(* CODESYS project GomelChemical.export

Project tree, tasks and I/O mapping:
  application Application
    libraries: 
    task PLC_Task (cyclic, interval t#50ms, priority 15) calls PLC_PRG
    GV/
      global variables _DO
      global variables AI
      global variables AO
      global variables DI
      global variables Hard
      global variables HMI_Sensors
      global variables HMI_Setting
    IO/
      function AI_TO_Current [ST]
      program prAItoValue [ST]
      program prInToVars [ST]
      program prVarsToOut [ST]
    program PLC_PRG [ST]
*)

// Application/GV/_DO

VAR_GLOBAL
	DO_SupplyStart_57_1	: BOOL;
	DO_SupplyStop_57_1	: BOOL;
	DO_SupplyStart_57_2	: BOOL;
	DO_SupplyStop_57_2	: BOOL;
	DO_SupplyStart_71_1	: BOOL;
	DO_SupplyStop_71_1	: BOOL;
	DO_SupplyStart_71_2	: BOOL;
	DO_SupplyStop_71_2	: BOOL;
	DO_SupplyStart_81_1	: BOOL;
	DO_SupplyStop_81_1	: BOOL;
	DO_MaxLevel_70_1_70_2_Stp_Elv8_Cvr5_6A:	BOOL;
	DO_MaxLevel_86_Stp_Elv8_Cvr5_7:	BOOL;
	DO_MinLevel_49_Stp_Pump_50:	BOOL;
	DO_MaxLevel_49_Stp_Pump_50:	BOOL;
	DO_MinLevel_67_Stp_Pump_68:	BOOL;
	DO_MaxLevel_67_Stp_Pump_68:	BOOL;
	DO_MinLevel_67_Stp_Pump_68_1:	BOOL;
	DO_MaxLevel_67_Stp_Pump_68_1:	BOOL;
	DO_MinLevel_103_1_Stp_Pump_103_1A:	BOOL;
	DO_MinLevelL1_103_1_Stp_Pump_103_1B:	BOOL;
	DO_MinLevelL2_103_1_Stp_Pump_103_1B:	BOOL;
	
//////////////////////////////////////////////////////////////////////	
	
	_DO_SupplyStart_57_1	: BOOL;
	_DO_SupplyStop_57_1	: BOOL;
	_DO_SupplyStart_57_2	: BOOL;
	_DO_SupplyStop_57_2	: BOOL;
	_DO_SupplyStart_71_1	: BOOL;
	_DO_SupplyStop_71_1	: BOOL;
	_DO_SupplyStart_71_2	: BOOL;
	_DO_SupplyStop_71_2	: BOOL;
	_DO_SupplyStart_81_1	: BOOL;
	_DO_SupplyStop_81_1	: BOOL;
	_DO_MaxLevel_70_1_70_2_Stp_Elv8_Cvr5_6A:	BOOL;
	_DO_MaxLevel_86_Stp_Elv8_Cvr5_7:	BOOL;
	_DO_MinLevel_49_Stp_Pump_50:	BOOL;
	_DO_MaxLevel_49_Stp_Pump_50:	BOOL;
	_DO_MinLevel_67_Stp_Pump_68:	BOOL;
	_DO_MaxLevel_67_Stp_Pump_68:	BOOL;
	_DO_MinLevel_67_Stp_Pump_68_1:	BOOL;
	_DO_MaxLevel_67_Stp_Pump_68_1:	BOOL;
	_DO_MinLevel_103_1_Stp_Pump_103_1A:	BOOL;
	_DO_MinLevelL1_103_1_Stp_Pump_103_1B:	BOOL;
	_DO_MinLevelL2_103_1_Stp_Pump_103_1B:	BOOL;
	
	
END_VAR

// Application/GV/AI

VAR_GLOBAL
	AI_TgasBeforeDryerDrum_45		: INT;
	AI_TgasAfterDryerDrum_45		: INT;
	AI_TgasFurnace_120				: INT;
	AI_TproductAfterDryerDrum_45	: INT;
	AI_TairCooler					: INT;
	AI_TairAfterDrumCond_76			: INT;
	AI_Tvent_53_3_1					: INT;
	AI_Tvent_53_3_2					: INT;
	AI_Tvent_53_2_1					: INT;
	AI_Tvent_53_2_2					: INT;
	AI_Tvent_53_1_1					: INT;
	AI_Tvent_53_1_2					: INT;
	
	AI_Tvent_65_0_1					: INT;
	AI_Tvent_65_0_2					: INT;
	AI_Tvent_65_1_1					: INT;
	AI_Tvent_65_1_2					: INT;
	AI_Tvent_65_2_1					: INT;
	AI_Tvent_65_2_2					: INT;
	AI_Tretur_61					: INT;
	AI_Ttank_103_1					: INT;
	AI_AirPressureBeforeBurner		: INT;
	AI_AirFirstPressureBeforeFurnace_120		: INT;
	AI_AirSecondPressureBeforeFurnace_120		: INT;
	AI_PCV22Pos						: INT;
	AI_UnderPresFurnace_120			: INT;
	AI_UnderPresGranul_31			: INT;
	AI_UnderPresDryerDrum_45		: INT;
	AI_UnderPresCooler_63_1			: INT;
	AI_PressureKiPA					: INT;
	AI_UnderPresBeforeAbsorbAKT_37	: INT;
	AI_UnderPresAfterAbsorbAKT_37	: INT;
	AI_UnderPresAfterAPS_48			: INT;
	AI_UnderPresBeforeHydroCycl_21	: INT;
	AI_UnderPresAfterHydroCycl_21	: INT;
	AI_UnderPresSalex_211			: INT;
	AI_AbsorbConsumInHydroCycl_21	: INT;
	AI_AbsorbConsumBeforeHydroCycl_21	: INT;
	AI_GasConsumBeforeBurner		: INT;
	AI_FCV16Pos						: INT;
	AI_AirConsumeFurnace_120		: INT;
	AI_FCV18Pos						: INT;
	AI_ReturConsumGranul_31			: INT;
	AI_AbsorLiquidConsumbAKT_37_FT100		: INT;
	AI_WaterConsumAbsorbSystem		: INT;
	AI_AbsorLiquidScuber_66_12		: INT;
	AI_AbsorLiquidTank_103_1		: INT;
	AI_FCV113						: INT;
	AI_ConsumBeforeScrubber_66_1	: INT;
	AI_ConsumInAPS_48				: INT;
	AI_ConsumH2SO4_102_to_35		: INT;
	AI_ConsumH2SO4_102_to_103		: INT;
	AI_AbsorLiquidConsumbAKT_37_FT132		: INT;
	AI_Consum_H3PO4					: INT;
	AI_ConsumH2SO4					: INT;
	AI_ConsumPressedAirToZech		: INT;
	AI_ConsumPressedAir				: INT;
	AI_ConsumChlKToGran_FQUIR_12_31	: INT;
	AI_ConsumKarbanToGran_31		: INT;
	AI_ConsumChlKToGran_FQUIR_17_31	: INT;
	AI_ConsumMicroAddToGran_31_FQUIR_57_1	: INT;
	AI_ConsumMicroAddToGran_31_FQUIR_57_2	: INT;
	AI_OilLevel_78					: INT;
	AI_CycleTankLevel_49			: INT;
	AI_LCV101Pos					: INT;
	AI_CollectorTankLevel_35		: INT;
	AI_CycleTankLevel_67			: INT;
	AI_CollectorTankLevel_103_1		: INT;
	AI_ReceivTankH3PO4level_41		: INT;
	AI_ReceivTankH3PO4level_39		: INT;
	AI_SupplyTankH3PO4level_25		: INT;
	AI_LCV203Pos					: INT;
	AI_TankH2SO4Level_102			: INT;
	AI_SupplyTankH2SO4Level_102_a	: INT;
	AI_LCV206Pos					: INT;
	AI_pH_CollectorTank_35			: INT;
	AI_ACV104Pos					: INT;
	AI_pH_CyclTank_49				: INT;
	AI_ACV112Pos					: INT;
	AI_pH_CollectorTank_103_1		: INT;
	AI_ACV115Pos					: INT;
	AI_OutAirWetness				: INT;
	AI_DryerRoomAirWetness_45			: INT;
	AI_IssuedProductWeight_203			: INT;
	AI_TubeReactorTemp_100_TE9			: INT;
	AI_AntiCackTempInReceiveTank_81	: INT;
	AI_TCV302Pos					: INT;
	AI_AntiCackTempInSupplyTank_81_TT303	: INT;
	AI_TCV303Pos					: INT;
	AI_TubeReactorTemp_100_TE304	: INT;
	AI_H2SO4_PressureBeforeTubeReactor_100	: INT;
	AI_H3PO4_PressureBeforeTubeReactor_100	: INT;
	AI_AcidWaistPressure_100				: INT;
	AI_H2SO4_PressureBeforeTubeReactor_100_1	: INT;
	AI_H3PO4_PressureBeforeTubeReactor_100_1	: INT;
	AI_AcidWaistPressure_100_1				: INT;
	AI_H2SO4ConsumTubeReactor_100		: INT;
	AI_FCV3Pos					: INT;
	AI_H3PO4ConsumTubeReactor_100		: INT;
	AI_FCV4Pos					: INT;
	AI_AcidWaistConsume_100				: INT;
	AI_FCV5Pos					: INT;
	AI_FCV10Pos					: INT;
	AI_FCV214Pos					: INT;
	AI_FCV341Pos					: INT;
	AI_FCV342Pos					: INT;
	AI_H2SO4ConsumTubeReactor_100_1		: INT;
	AI_FCV343Pos					: INT;
	AI_H3PO4ConsumTubeReactor_100_1		: INT;
	AI_FCV344Pos					: INT;
	AI_AcidWaistConsume_100_1		: INT;
	AI_FCV345Pos					: INT;
	AI_FCV346Pos					: INT;
	AI_AntiCackLevelInReceivTank_81	: INT;
	AI_AntiCackLevelInSupplyTank_82	: INT;
	AI_SubPumpCurrent_102_B				: INT;
	AI_SubPumpCurrent_103_1B		: INT;
	
	
	
	//////////////////////////////////////////////////////////////////
	
	_AI_TgasBeforeDryerDrum_45		: INT;
	_AI_TgasAfterDryerDrum_45		: INT;
	_AI_TgasFurnace_120				: INT;
	_AI_TproductAfterDryerDrum_45	: INT;
	_AI_TairCooler					: INT;
	_AI_TairAfterDrumCond_76			: INT;
	_AI_Tvent_53_3_1					: INT;
	_AI_Tvent_53_3_2					: INT;
	_AI_Tvent_53_2_1					: INT;
	_AI_Tvent_53_2_2					: INT;
	_AI_Tvent_53_1_1					: INT;
	_AI_Tvent_53_1_2					: INT;
	
	_AI_Tvent_65_0_1					: INT;
	_AI_Tvent_65_0_2					: INT;
	_AI_Tvent_65_1_1					: INT;
	_AI_Tvent_65_1_2					: INT;
	_AI_Tvent_65_2_1					: INT;
	_AI_Tvent_65_2_2					: INT;
	_AI_Tretur_61					: INT;
	_AI_Ttank_103_1					: INT;
	_AI_AirPressureBeforeBurner		: INT;
	_AI_AirFirstPressureBeforeFurnace_120		: INT;
	_AI_AirSecondPressureBeforeFurnace_120		: INT;
	_AI_PCV22Pos						: INT;
	_AI_UnderPresFurnace_120			: INT;
	_AI_UnderPresGranul_31			: INT;
	_AI_UnderPresDryerDrum_45		: INT;
	_AI_UnderPresCooler_63_1			: INT;
	_AI_PressureKiPA					: INT;
	_AI_UnderPresBeforeAbsorbAKT_37	: INT;
	_AI_UnderPresAfterAbsorbAKT_37	: INT;
	_AI_UnderPresAfterAPS_48			: INT;
	_AI_UnderPresBeforeHydroCycl_21	: INT;
	_AI_UnderPresAfterHydroCycl_21	: INT;
	_AI_UnderPresSalex_211			: INT;
	_AI_AbsorbConsumInHydroCycl_21	: INT;
	_AI_AbsorbConsumBeforeHydroCycl_21	: INT;
	_AI_GasConsumBeforeBurner		: INT;
	_AI_FCV16Pos						: INT;
	_AI_AirConsumeFurnace_120		: INT;
	_AI_FCV18Pos						: INT;
	_AI_ReturConsumGranul_31			: INT;
	_AI_AbsorLiquidConsumbAKT_37_FT100		: INT;
	_AI_WaterConsumAbsorbSystem		: INT;
	_AI_AbsorLiquidScuber_66_12		: INT;
	_AI_AbsorLiquidTank_103_1		: INT;
	_AI_FCV113						: INT;
	_AI_ConsumBeforeScrubber_66_1	: INT;
	_AI_ConsumInAPS_48				: INT;
	_AI_ConsumH2SO4_102_to_35		: INT;
	_AI_ConsumH2SO4_102_to_103		: INT;
	_AI_AbsorLiquidConsumbAKT_37_FT132		: INT;
	_AI_Consum_H3PO4					: INT;
	_AI_ConsumH2SO4					: INT;
	_AI_ConsumPressedAirToZech		: INT;
	_AI_ConsumPressedAir				: INT;
	_AI_ConsumChlKToGran_FQUIR_12_31	: INT;
	_AI_ConsumKarbanToGran_31		: INT;
	_AI_ConsumChlKToGran_FQUIR_17_31	: INT;
	_AI_ConsumMicroAddToGran_31_FQUIR_57_1	: INT;
	_AI_ConsumMicroAddToGran_31_FQUIR_57_2	: INT;
	_AI_OilLevel_78					: INT;
	_AI_CycleTankLevel_49			: INT;
	_AI_LCV101Pos					: INT;
	_AI_CollectorTankLevel_35		: INT;
	_AI_CycleTankLevel_67			: INT;
	_AI_CollectorTankLevel_103_1		: INT;
	_AI_ReceivTankH3PO4level_41		: INT;
	_AI_ReceivTankH3PO4level_39		: INT;
	_AI_SupplyTankH3PO4level_25		: INT;
	_AI_LCV203Pos					: INT;
	_AI_TankH2SO4Level_102			: INT;
	_AI_SupplyTankH2SO4Level_102_a	: INT;
	_AI_LCV206Pos					: INT;
	_AI_pH_CollectorTank_35			: INT;
	_AI_ACV104Pos					: INT;
	_AI_pH_CyclTank_49				: INT;
	_AI_ACV112Pos					: INT;
	_AI_pH_CollectorTank_103_1		: INT;
	_AI_ACV115Pos					: INT;
	_AI_OutAirWetness				: INT;
	_AI_DryerRoomAirWetness_45			: INT;
	_AI_IssuedProductWeight_203			: INT;
	_AI_TubeReactorTemp_100_TE9			: INT;
	_AI_AntiCackTempInReceiveTank_81	: INT;
	_AI_TCV302Pos					: INT;
	_AI_AntiCackTempInSupplyTank_81_TT303	: INT;
	_AI_TCV303Pos					: INT;
	_AI_TubeReactorTemp_100_TE304	: INT;
	_AI_H2SO4_PressureBeforeTubeReactor_100	: INT;
	_AI_H3PO4_PressureBeforeTubeReactor_100	: INT;
	_AI_AcidWaistPressure_100				: INT;
	_AI_H2SO4_PressureBeforeTubeReactor_100_1	: INT;
	_AI_H3PO4_PressureBeforeTubeReactor_100_1	: INT;
	_AI_AcidWaistPressure_100_1				: INT;
	_AI_H2SO4ConsumTubeReactor_100		: INT;
	_AI_FCV3Pos					: INT;
	_AI_H3PO4ConsumTubeReactor_100		: INT;
	_AI_FCV4Pos					: INT;
	_AI_AcidWaistConsume_100				: INT;
	_AI_FCV5Pos					: INT;
	_AI_FCV10Pos					: INT;
	_AI_FCV214Pos					: INT;
	_AI_FCV341Pos					: INT;
	_AI_FCV342Pos					: INT;
	_AI_H2SO4ConsumTubeReactor_100_1		: INT;
	_AI_FCV343Pos					: INT;
	_AI_H3PO4ConsumTubeReactor_100_1		: INT;
	_AI_FCV344Pos					: INT;
	_AI_AcidWaistConsume_100_1		: INT;
	_AI_FCV345Pos					: INT;
	_AI_FCV346Pos					: INT;
	_AI_AntiCackLevelInReceivTank_81	: INT;
	_AI_AntiCackLevelInSupplyTank_82	: INT;
	_AI_SubPumpCurrent_102_B				: INT;
	_AI_SubPumpCurrent_103_1B		: INT;
	
	
	
	
	
	
	
	
	
			
END_VAR

// Application/GV/AO

VAR_GLOBAL
	AO_AirPressureBeforeFenese_120		: INT;
	AO_GasFlowBeforeBurner				: INT;
	AO_AirFlowFenese_120				: INT;
	AO_AbsorbLiquidTo_103_1				: INT;
	AO_ChlorKFlowToGranul_31_FQIR12		: INT;
	AO_KarbonFlowToGranul_31			: INT;
	AO_ChlorKFlowToGranul_31_FQIR17		: INT;
	AO_MicroAddToGranul_31_FQIR57_1		: INT;
	AO_MicroAddToGranul_31_FQIR57_2		: INT;
	AO_SetLevelCyclTank_49				: INT;
	AO_SetLevelH3PO4SupplyTank_25		: INT;
	AO_SetLevelH2SO4SupplyTank_102_a	: INT;
	AO_Set_pHCollectTank_35				: INT;
	AO_Set_pHCycleTank_49				: INT;
	AO_Set_pHCollectTank_103_1			: INT;
	AO_SetShyberVent_53_3				: INT;
	AO_SetShyberVent_53_2				: INT;
	AO_SetShyberVent_53_1				: INT;
	AO_SetShyberVent_65_0				: INT;
	AO_SetShyberVent_65_1				: INT;
	AO_SetShyberVent_65_2				: INT;
	AO_SetAntiCackTempInCollectTank_81	: INT;
	AO_SetAntiCackTempInCollectTank_82	: INT;
	AO_SetH2SO4SupplyToTubeReactor_100	: INT;
	AO_SetH3PO4SupplyToTubeReactor_100	: INT;
	AO_SetAcidWaistFlowToTubeReactor_100	: INT;
	AO_SetNH3FlowToTubeReactor_100		: INT;
	AO_SetSteamFlowToTubeReactor_100	: INT;
	AO_SetAntiCackFlawToCondDrum_76		: INT;
	AO_SetNH3FlowToTubeReactor_100_1	: INT;
	AO_SetH2SO4SupplyToTubeReactor_100_1	: INT;
	AO_SetH3PO4SupplyToTubeReactor_100_1	: INT;
	AO_SetAcidWaistFlowToTubeReactor_100_1	: INT;
	AO_SetSteamFlowToTubeReactor_100_1	: INT;
	
	
	
	
	/////////////////////////////////////////////////////////////////////
	
	
	
	_AO_AirPressureBeforeFenese_120		: INT;
	_AO_GasFlowBeforeBurner				: INT;
	_AO_AirFlowFenese_120				: INT;
	_AO_AbsorbLiquidTo_103_1				: INT;
	_AO_ChlorKFlowToGranul_31_FQIR12		: INT;
	_AO_KarbonFlowToGranul_31			: INT;
	_AO_ChlorKFlowToGranul_31_FQIR17		: INT;
	_AO_MicroAddToGranul_31_FQIR57_1		: INT;
	_AO_MicroAddToGranul_31_FQIR57_2		: INT;
	_AO_SetLevelCyclTank_49				: INT;
	_AO_SetLevelH3PO4SupplyTank_25		: INT;
	_AO_SetLevelH2SO4SupplyTank_102_a	: INT;
	_AO_Set_pHCollectTank_35				: INT;
	_AO_Set_pHCycleTank_49				: INT;
	_AO_Set_pHCollectTank_103_1			: INT;
	_AO_SetShyberVent_53_3				: INT;
	_AO_SetShyberVent_53_2				: INT;
	_AO_SetShyberVent_53_1				: INT;
	_AO_SetShyberVent_65_0				: INT;
	_AO_SetShyberVent_65_1				: INT;
	_AO_SetShyberVent_65_2				: INT;
	_AO_SetAntiCackTempInCollectTank_81	: INT;
	_AO_SetAntiCackTempInCollectTank_82	: INT;
	_AO_SetH2SO4SupplyToTubeReactor_100	: INT;
	_AO_SetH3PO4SupplyToTubeReactor_100	: INT;
	_AO_SetAcidWaistFlowToTubeReactor_100	: INT;
	_AO_SetNH3FlowToTubeReactor_100		: INT;
	_AO_SetSteamFlowToTubeReactor_100	: INT;
	_AO_SetAntiCackFlawToCondDrum_76		: INT;
	_AO_SetNH3FlowToTubeReactor_100_1	: INT;
	_AO_SetH2SO4SupplyToTubeReactor_100_1	: INT;
	_AO_SetH3PO4SupplyToTubeReactor_100_1	: INT;
	_AO_SetAcidWaistFlowToTubeReactor_100_1	: INT;
	_AO_SetSteamFlowToTubeReactor_100_1	: INT;
	
	
	
END_VAR

// Application/GV/DI

VAR_GLOBAL
	DI_GasFurnaceMinLevelAlm			: BOOL;
	DI_BunkerMaxLevel_88_2				: BOOL;
	DI_BunkerMaxLevel_88_1				: BOOL;
	DI_BunkerMaxLevel_70_1				: BOOL;
	DI_BunkerMaxLevel_70_2				: BOOL;
	DI_BunkerMaxLevel_86				: BOOL;
	DI_ElevatorMaxLevel_54				: BOOL;
	DI_OvenMaxLevel_58_1				: BOOL;
	DI_ElevatorMaxLevel_214_1			: BOOL;
	DI_MainBurnerFire_120				: BOOL;
	DI_IgnitionBurnerFire_120			: BOOL;
	DI_SupplierMotorWork_57_1			: BOOL;
	DI_SupplierMotorAlm_57_1			: BOOL;
	DI_SupplierMotorWork_57_2			: BOOL;
	DI_SupplierMotorAlm_57_2			: BOOL;
	DI_SupplierMotorWork_71_1			: BOOL;
	DI_SupplierMotorAlm_71_1			: BOOL;
	DI_SupplierMotorWork_71_2			: BOOL;
	DI_SupplierMotorAlm_71_2			: BOOL;
	DI_SupplierMotorWork_87_1			: BOOL;
	DI_SupplierMotorAlm_87_1			: BOOL;
	DI_DryerDrumMotorNotWorking_45_53	: BOOL;
	DI_UPS_Bypass_1						: BOOL;
	DI_UPS_Battery_1					: BOOL;
	DI_UPS_BatteryDischarge_1			: BOOL;
	DI_UPS_Alm_1						: BOOL;
	DI_UPS_Bypass_2						: BOOL;
	DI_UPS_Battery_2					: BOOL;
	DI_UPS_BatteryDischarge_2			: BOOL;
	DI_UPS_Alm_2						: BOOL;
	DI_PowerRackVoltageOn_1				: BOOL;
	DI_PowerRackVoltageOn_2				: BOOL;
	DI_PowerRackAlmStop_1				: BOOL;
	DI_PowerRackAlmStop_2				: BOOL;
	DI_SubPumpWorking_25_1B				: BOOL;
	DI_AntiCackPumpWorking_81_1			: BOOL;
	DI_AntiCackPumpWorking_81_2			: BOOL;
	DI_AntiCackPumpWorking_82_1			: BOOL;
	DI_AntiCackPumpWorking_82_2			: BOOL;
	DI_SubPumpWorking_102_B				: BOOL;
	
	
	
	///////////////////////////////////////////////////////////////////////////
	
	
	_DI_GasFurnaceMinLevelAlm			: BOOL;
	_DI_BunkerMaxLevel_88_2				: BOOL;
	_DI_BunkerMaxLevel_88_1				: BOOL;
	_DI_BunkerMaxLevel_70_1				: BOOL;
	_DI_BunkerMaxLevel_70_2				: BOOL;
	_DI_BunkerMaxLevel_86				: BOOL;
	_DI_ElevatorMaxLevel_54				: BOOL;
	_DI_OvenMaxLevel_58_1				: BOOL;
	_DI_ElevatorMaxLevel_214_1			: BOOL;
	_DI_MainBurnerFire_120				: BOOL;
	_DI_IgnitionBurnerFire_120			: BOOL;
	_DI_SupplierMotorWork_57_1			: BOOL;
	_DI_SupplierMotorAlm_57_1			: BOOL;
	_DI_SupplierMotorWork_57_2			: BOOL;
	_DI_SupplierMotorAlm_57_2			: BOOL;
	_DI_SupplierMotorWork_71_1			: BOOL;
	_DI_SupplierMotorAlm_71_1			: BOOL;
	_DI_SupplierMotorWork_71_2			: BOOL;
	_DI_SupplierMotorAlm_71_2			: BOOL;
	_DI_SupplierMotorWork_87_1			: BOOL;
	_DI_SupplierMotorAlm_87_1			: BOOL;
	_DI_DryerDrumMotorNotWorking_45_53	: BOOL;
	_DI_UPS_Bypass_1						: BOOL;
	_DI_UPS_Battery_1					: BOOL;
	_DI_UPS_BatteryDischarge_1			: BOOL;
	_DI_UPS_Alm_1						: BOOL;
	_DI_UPS_Bypass_2						: BOOL;
	_DI_UPS_Battery_2					: BOOL;
	_DI_UPS_BatteryDischarge_2			: BOOL;
	_DI_UPS_Alm_2						: BOOL;
	_DI_PowerRackVoltageOn_1				: BOOL;
	_DI_PowerRackVoltageOn_2				: BOOL;
	_DI_PowerRackAlmStop_1				: BOOL;
	_DI_PowerRackAlmStop_2				: BOOL;
	_DI_SubPumpWorking_25_1B				: BOOL;
	_DI_AntiCackPumpWorking_81_1			: BOOL;
	_DI_AntiCackPumpWorking_81_2			: BOOL;
	_DI_AntiCackPumpWorking_82_1			: BOOL;
	_DI_AntiCackPumpWorking_82_2			: BOOL;
	_DI_SubPumpWorking_102_B				: BOOL;
	
	
	
	
	
END_VAR

// Application/GV/Hard

VAR_GLOBAL
	AI_OilConsumeBeforeDrumCond_76	: REAL;
	AI_OilTempBeforeDrumCond_76		: REAL;
	AI_OilDensBeforeDrumCond_76		: REAL;
	AI_SteamConsume					: REAL;
	AI_SteamTemp					: REAL;
	AI_SteamPress					: REAL;
	AI_NH3_TubeReactConsume_100		: REAL;
	AI_NH3_TubeReactDens_100		: REAL;
	AI_NH3_TubeReactTemp_100		: REAL;
	AI_SteamTubeReactConsume_100		: REAL;
	AI_SteamTubeReactTemp_100			: REAL;
	AI_SteamTubeReactPress_100			: REAL;
	AI_AntiCackCondDrumConsume		: REAL;
	AI_NH3_TubeReactConsume_100_1	: REAL;
	AI_NH3_TubeReactDens_100_1		: REAL;
	AI_NH3_TubeReactTemp_100_1		: REAL;
	AI_SteamTubeReactConsume_100_1		: REAL;
	AI_SteamTubeReactTemp_100_1			: REAL;
	AI_SteamTubeReactPress_100_1			: REAL;
	
END_VAR

// Application/GV/HMI_Sensors

VAR_GLOBAL
TgasBeforeDryerDrum_45				:	REAL;
TgasAfterDryerDrum_45				:	REAL;
TgasFurnace_120						:	REAL;
TproductAfterDryerDrum_45			:	REAL;
TairCooler							:	REAL;
TairAfterDrumCond_76				:	REAL;
Tvent_53_3_1						:	REAL;
Tvent_53_3_2						:	REAL;
Tvent_53_2_1						:	REAL;
Tvent_53_2_2						:	REAL;
Tvent_53_1_1						:	REAL;
Tvent_53_1_2						:	REAL;
Tvent_65_0_1						:	REAL;
Tvent_65_0_2						:	REAL;
Tvent_65_1_1						:	REAL;
Tvent_65_1_2						:	REAL;
Tvent_65_2_1						:	REAL;
Tvent_65_2_2						:	REAL;
Tretur_61							:	REAL;
Ttank_103_1							:	REAL;
AirPressureBeforeBurner				:	REAL;
AirFirstPressureBeforeFurnace_120	:	REAL;
AirSecondPressureBeforeFurnace_120	:	REAL;
PCV22Pos							:	REAL;
UnderPresFurnace_120				:	REAL;
UnderPresGranul_31					:	REAL;
UnderPresDryerDrum_45				:	REAL;
UnderPresCooler_63_1				:	REAL;
PressureKiPA						:	REAL;
UnderPresBeforeAbsorbAKT_37			:	REAL;
UnderPresAfterAbsorbAKT_37			:	REAL;
UnderPresAfterAPS_48				:	REAL;
UnderPresBeforeHydroCycl_21			:	REAL;
UnderPresAfterHydroCycl_21			:	REAL;
UnderPresSalex_211					:	REAL;
AbsorbConsumInHydroCycl_21			:	REAL;
AbsorbConsumBeforeHydroCycl_21		:	REAL;
GasConsumBeforeBurner				:	REAL;
FCV16Pos							:	REAL;
AirConsumeFurnace_120				:	REAL;
FCV18Pos							:	REAL;
ReturConsumGranul_31				:	REAL;
AbsorLiquidConsumbAKT_37_FT100		:	REAL;
WaterConsumAbsorbSystem				:	REAL;
AbsorLiquidScuber_66_12				:	REAL;
AbsorLiquidTank_103_1				:	REAL;
FCV113								:	REAL;
ConsumBeforeScrubber_66_1			:	REAL;
ConsumInAPS_48						:	REAL;
ConsumH2SO4_102_to_35				:	REAL;
ConsumH2SO4_102_to_103				:	REAL;
AbsorLiquidConsumbAKT_37_FT132		:	REAL;
Consum_H3PO4						:	REAL;
ConsumH2SO4							:	REAL;
ConsumPressedAirToZech				:	REAL;
ConsumPressedAir					:	REAL;
ConsumChlKToGran_FQUIR_12_31		:	REAL;
ConsumKarbanToGran_31				:	REAL;
ConsumChlKToGran_FQUIR_17_31		:	REAL;
ConsumMicroAddToGran_31_FQUIR_57_1	:	REAL;
ConsumMicroAddToGran_31_FQUIR_57_2	:	REAL;
OilLevel_78							:	REAL;
CycleTankLevel_49					:	REAL;
LCV101Pos							:	REAL;
CollectorTankLevel_35				:	REAL;
CycleTankLevel_67					:	REAL;
CollectorTankLevel_103_1			:	REAL;
ReceivTankH3PO4level_41				:	REAL;
ReceivTankH3PO4level_39				:	REAL;
SupplyTankH3PO4level_25				:	REAL;
LCV203Pos							:	REAL;
TankH2SO4Level_102					:	REAL;
SupplyTankH2SO4Level_102_a			:	REAL;
LCV206Pos							:	REAL;
pH_CollectorTank_35					:	REAL;
ACV104Pos							:	REAL;
pH_CyclTank_49						:	REAL;
ACV112Pos							:	REAL;
pH_CollectorTank_103_1				:	REAL;
ACV115Pos							:	REAL;
OutAirWetness						:	REAL;
DryerRoomAirWetness_45				:	REAL;
IssuedProductWeight_203				:	REAL;
TubeReactorTemp_100_TE9				:	REAL;
AntiCackTempInReceiveTank_81		:	REAL;
TCV302Pos							:	REAL;
AntiCackTempInSupplyTank_81_TT303	:	REAL;
TCV303Pos							:	REAL;
TubeReactorTemp_100_TE304			:	REAL;
H2SO4_PressureBeforeTubeReactor_100	:	REAL;
H3PO4_PressureBeforeTubeReactor_100	:	REAL;
AcidWaistPressure_100				:	REAL;
H2SO4_PressureBeforeTubeReactor_100_1	:	REAL;
H3PO4_PressureBeforeTubeReactor_100_1	:	REAL;
AcidWaistPressure_100_1				:	REAL;
H2SO4ConsumTubeReactor_100			:	REAL;
FCV3Pos								:	REAL;
H3PO4ConsumTubeReactor_100			:	REAL;
FCV4Pos								:	REAL;
AcidWaistConsume_100				:	REAL;
FCV5Pos								:	REAL;
FCV10Pos							:	REAL;
FCV214Pos							:	REAL;
FCV341Pos							:	REAL;
FCV342Pos							:	REAL;
H2SO4ConsumTubeReactor_100_1		:	REAL;
FCV343Pos							:	REAL;
H3PO4ConsumTubeReactor_100_1		:	REAL;
FCV344Pos							:	REAL;
AcidWaistConsume_100_1				:	REAL;
FCV345Pos							:	REAL;
FCV346Pos							:	REAL;
AntiCackLevelInReceivTank_81		:	REAL;
AntiCackLevelInSupplyTank_82		:	REAL;
SubPumpCurrent_102_B				:	REAL;
SubPumpCurrent_103_1B				:	REAL;


END_VAR

// Application/GV/HMI_Setting

VAR_GLOBAL
TgasBeforeDryerDrum_45_CalCoef				:	REAL:=1;
TgasAfterDryerDrum_45_CalCoef				:	REAL:=1;
TgasFurnace_120_CalCoef				:	REAL:=1;
TproductAfterDryerDrum_45_CalCoef				:	REAL:=1;
TairCooler_CalCoef				:	REAL:=1;
TairAfterDrumCond_76_CalCoef				:	REAL:=1;
Tvent_53_3_1_CalCoef				:	REAL:=1;
Tvent_53_3_2_CalCoef				:	REAL:=1;
Tvent_53_2_1_CalCoef				:	REAL:=1;
Tvent_53_2_2_CalCoef				:	REAL:=1;
Tvent_53_1_1_CalCoef				:	REAL:=1;
Tvent_53_1_2_CalCoef				:	REAL:=1;
Tvent_65_0_1_CalCoef				:	REAL:=1;
Tvent_65_0_2_CalCoef				:	REAL:=1;
Tvent_65_1_1_CalCoef				:	REAL:=1;
Tvent_65_1_2_CalCoef				:	REAL:=1;
Tvent_65_2_1_CalCoef				:	REAL:=1;
Tvent_65_2_2_CalCoef				:	REAL:=1;
Tretur_61_CalCoef				:	REAL:=1;
Ttank_103_1_CalCoef				:	REAL:=1;
AirPressureBeforeBurner_CalCoef				:	REAL:=1;
AirFirstPressureBeforeFurnace_120_CalCoef				:	REAL:=1;
AirSecondPressureBeforeFurnace_120_CalCoef				:	REAL:=1;
PCV22Pos_CalCoef				:	REAL:=1;
UnderPresFurnace_120_CalCoef				:	REAL:=1;
UnderPresGranul_31_CalCoef				:	REAL:=1;
UnderPresDryerDrum_45_CalCoef				:	REAL:=1;
UnderPresCooler_63_1_CalCoef				:	REAL:=1;
PressureKiPA_CalCoef				:	REAL:=1;
UnderPresBeforeAbsorbAKT_37_CalCoef				:	REAL:=1;
UnderPresAfterAbsorbAKT_37_CalCoef				:	REAL:=1;
UnderPresAfterAPS_48_CalCoef				:	REAL:=1;
UnderPresBeforeHydroCycl_21_CalCoef				:	REAL:=1;
UnderPresAfterHydroCycl_21_CalCoef				:	REAL:=1;
UnderPresSalex_211_CalCoef				:	REAL:=1;
AbsorbConsumInHydroCycl_21_CalCoef				:	REAL:=1;
AbsorbConsumBeforeHydroCycl_21_CalCoef				:	REAL:=1;
GasConsumBeforeBurner_CalCoef				:	REAL:=1;
FCV16Pos_CalCoef				:	REAL:=1;
AirConsumeFurnace_120_CalCoef				:	REAL:=1;
FCV18Pos_CalCoef				:	REAL:=1;
ReturConsumGranul_31_CalCoef				:	REAL:=1;
AbsorLiquidConsumbAKT_37_FT100_CalCoef				:	REAL:=1;
WaterConsumAbsorbSystem_CalCoef				:	REAL:=1;
AbsorLiquidScuber_66_12_CalCoef				:	REAL:=1;
AbsorLiquidTank_103_1_CalCoef				:	REAL:=1;
FCV113_CalCoef				:	REAL:=1;
ConsumBeforeScrubber_66_1_CalCoef				:	REAL:=1;
ConsumInAPS_48_CalCoef				:	REAL:=1;
ConsumH2SO4_102_to_35_CalCoef				:	REAL:=1;
ConsumH2SO4_102_to_103_CalCoef				:	REAL:=1;
AbsorLiquidConsumbAKT_37_FT132_CalCoef				:	REAL:=1;
Consum_H3PO4_CalCoef				:	REAL:=1;
ConsumH2SO4_CalCoef				:	REAL:=1;
ConsumPressedAirToZech_CalCoef				:	REAL:=1;
ConsumPressedAir_CalCoef				:	REAL:=1;
ConsumChlKToGran_FQUIR_12_31_CalCoef				:	REAL:=1;
ConsumKarbanToGran_31_CalCoef				:	REAL:=1;
ConsumChlKToGran_FQUIR_17_31_CalCoef				:	REAL:=1;
ConsumMicroAddToGran_31_FQUIR_57_1_CalCoef				:	REAL:=1;
ConsumMicroAddToGran_31_FQUIR_57_2_CalCoef				:	REAL:=1;
OilLevel_78_CalCoef				:	REAL:=1;
CycleTankLevel_49_CalCoef				:	REAL:=1;
LCV101Pos_CalCoef				:	REAL:=1;
CollectorTankLevel_35_CalCoef				:	REAL:=1;
CycleTankLevel_67_CalCoef				:	REAL:=1;
CollectorTankLevel_103_1_CalCoef				:	REAL:=1;
ReceivTankH3PO4level_41_CalCoef				:	REAL:=1;
ReceivTankH3PO4level_39_CalCoef				:	REAL:=1;
SupplyTankH3PO4level_25_CalCoef				:	REAL:=1;
LCV203Pos_CalCoef				:	REAL:=1;
TankH2SO4Level_102_CalCoef				:	REAL:=1;
SupplyTankH2SO4Level_102_a_CalCoef				:	REAL:=1;
LCV206Pos_CalCoef				:	REAL:=1;
pH_CollectorTank_35_CalCoef				:	REAL:=1;
ACV104Pos_CalCoef				:	REAL:=1;
pH_CyclTank_49_CalCoef				:	REAL:=1;
ACV112Pos_CalCoef				:	REAL:=1;
pH_CollectorTank_103_1_CalCoef				:	REAL:=1;
ACV115Pos_CalCoef				:	REAL:=1;
OutAirWetness_CalCoef				:	REAL:=1;
DryerRoomAirWetness_45_CalCoef				:	REAL:=1;
IssuedProductWeight_203_CalCoef				:	REAL:=1;
TubeReactorTemp_100_TE9_CalCoef				:	REAL:=1;
AntiCackTempInReceiveTank_81_CalCoef				:	REAL:=1;
TCV302Pos_CalCoef				:	REAL:=1;
AntiCackTempInSupplyTank_81_TT303_CalCoef				:	REAL:=1;
TCV303Pos_CalCoef				:	REAL:=1;
TubeReactorTemp_100_TE304_CalCoef				:	REAL:=1;
H2SO4_PressureBeforeTubeReactor_100_CalCoef				:	REAL:=1;
H3PO4_PressureBeforeTubeReactor_100_CalCoef				:	REAL:=1;
AcidWaistPressure_100_CalCoef				:	REAL:=1;
H2SO4_PressureBeforeTubeReactor_100_1_CalCoef				:	REAL:=1;
H3PO4_PressureBeforeTubeReactor_100_1_CalCoef				:	REAL:=1;
AcidWaistPressure_100_1_CalCoef				:	REAL:=1;
H2SO4ConsumTubeReactor_100_CalCoef				:	REAL:=1;
FCV3Pos_CalCoef				:	REAL:=1;
H3PO4ConsumTubeReactor_100_CalCoef				:	REAL:=1;
FCV4Pos_CalCoef				:	REAL:=1;
AcidWaistConsume_100_CalCoef				:	REAL:=1;
FCV5Pos_CalCoef				:	REAL:=1;
FCV10Pos_CalCoef				:	REAL:=1;
FCV214Pos_CalCoef				:	REAL:=1;
FCV341Pos_CalCoef				:	REAL:=1;
FCV342Pos_CalCoef				:	REAL:=1;
H2SO4ConsumTubeReactor_100_1_CalCoef				:	REAL:=1;
FCV343Pos_CalCoef				:	REAL:=1;
H3PO4ConsumTubeReactor_100_1_CalCoef				:	REAL:=1;
FCV344Pos_CalCoef				:	REAL:=1;
AcidWaistConsume_100_1_CalCoef				:	REAL:=1;
FCV345Pos_CalCoef				:	REAL:=1;
FCV346Pos_CalCoef				:	REAL:=1;
AntiCackLevelInReceivTank_81_CalCoef				:	REAL:=1;
AntiCackLevelInSupplyTank_82_CalCoef				:	REAL:=1;
SubPumpCurrent_102_B_CalCoef				:	REAL:=1;
SubPumpCurrent_103_1B_CalCoef				:	REAL:=1;


////////////////////////////////////////////////////////////////////////////////////////////////////


TgasBeforeDryerDrum_45_Offset				:	REAL;
TgasAfterDryerDrum_45_Offset				:	REAL;
TgasFurnace_120_Offset				:	REAL;
TproductAfterDryerDrum_45_Offset				:	REAL;
TairCooler_Offset				:	REAL;
TairAfterDrumCond_76_Offset				:	REAL;
Tvent_53_3_1_Offset				:	REAL;
Tvent_53_3_2_Offset				:	REAL;
Tvent_53_2_1_Offset				:	REAL;
Tvent_53_2_2_Offset				:	REAL;
Tvent_53_1_1_Offset				:	REAL;
Tvent_53_1_2_Offset				:	REAL;
Tvent_65_0_1_Offset				:	REAL;
Tvent_65_0_2_Offset				:	REAL;
Tvent_65_1_1_Offset				:	REAL;
Tvent_65_1_2_Offset				:	REAL;
Tvent_65_2_1_Offset				:	REAL;
Tvent_65_2_2_Offset				:	REAL;
Tretur_61_Offset				:	REAL;
Ttank_103_1_Offset				:	REAL;
AirPressureBeforeBurner_Offset				:	REAL;
AirFirstPressureBeforeFurnace_120_Offset				:	REAL;
AirSecondPressureBeforeFurnace_120_Offset				:	REAL;
PCV22Pos_Offset				:	REAL;
UnderPresFurnace_120_Offset				:	REAL;
UnderPresGranul_31_Offset				:	REAL;
UnderPresDryerDrum_45_Offset				:	REAL;
UnderPresCooler_63_1_Offset				:	REAL;
PressureKiPA_Offset				:	REAL;
UnderPresBeforeAbsorbAKT_37_Offset				:	REAL;
UnderPresAfterAbsorbAKT_37_Offset				:	REAL;
UnderPresAfterAPS_48_Offset				:	REAL;
UnderPresBeforeHydroCycl_21_Offset				:	REAL;
UnderPresAfterHydroCycl_21_Offset				:	REAL;
UnderPresSalex_211_Offset				:	REAL;
AbsorbConsumInHydroCycl_21_Offset				:	REAL;
AbsorbConsumBeforeHydroCycl_21_Offset				:	REAL;
GasConsumBeforeBurner_Offset				:	REAL;
FCV16Pos_Offset				:	REAL;
AirConsumeFurnace_120_Offset				:	REAL;
FCV18Pos_Offset				:	REAL;
ReturConsumGranul_31_Offset				:	REAL;
AbsorLiquidConsumbAKT_37_FT100_Offset				:	REAL;
WaterConsumAbsorbSystem_Offset				:	REAL;
AbsorLiquidScuber_66_12_Offset				:	REAL;
AbsorLiquidTank_103_1_Offset				:	REAL;
FCV113_Offset				:	REAL;
ConsumBeforeScrubber_66_1_Offset				:	REAL;
ConsumInAPS_48_Offset				:	REAL;
ConsumH2SO4_102_to_35_Offset				:	REAL;
ConsumH2SO4_102_to_103_Offset				:	REAL;
AbsorLiquidConsumbAKT_37_FT132_Offset				:	REAL;
Consum_H3PO4_Offset				:	REAL;
ConsumH2SO4_Offset				:	REAL;
ConsumPressedAirToZech_Offset				:	REAL;
ConsumPressedAir_Offset				:	REAL;
ConsumChlKToGran_FQUIR_12_31_Offset				:	REAL;
ConsumKarbanToGran_31_Offset				:	REAL;
ConsumChlKToGran_FQUIR_17_31_Offset				:	REAL;
ConsumMicroAddToGran_31_FQUIR_57_1_Offset				:	REAL;
ConsumMicroAddToGran_31_FQUIR_57_2_Offset				:	REAL;
OilLevel_78_Offset				:	REAL;
CycleTankLevel_49_Offset				:	REAL;
LCV101Pos_Offset				:	REAL;
CollectorTankLevel_35_Offset				:	REAL;
CycleTankLevel_67_Offset				:	REAL;
CollectorTankLevel_103_1_Offset				:	REAL;
ReceivTankH3PO4level_41_Offset				:	REAL;
ReceivTankH3PO4level_39_Offset				:	REAL;
SupplyTankH3PO4level_25_Offset				:	REAL;
LCV203Pos_Offset				:	REAL;
TankH2SO4Level_102_Offset				:	REAL;
SupplyTankH2SO4Level_102_a_Offset				:	REAL;
LCV206Pos_Offset				:	REAL;
pH_CollectorTank_35_Offset				:	REAL;
ACV104Pos_Offset				:	REAL;
pH_CyclTank_49_Offset				:	REAL;
ACV112Pos_Offset				:	REAL;
pH_CollectorTank_103_1_Offset				:	REAL;
ACV115Pos_Offset				:	REAL;
OutAirWetness_Offset				:	REAL;
DryerRoomAirWetness_45_Offset				:	REAL;
IssuedProductWeight_203_Offset				:	REAL;
TubeReactorTemp_100_TE9_Offset				:	REAL;
AntiCackTempInReceiveTank_81_Offset				:	REAL;
TCV302Pos_Offset				:	REAL;
AntiCackTempInSupplyTank_81_TT303_Offset				:	REAL;
TCV303Pos_Offset				:	REAL;
TubeReactorTemp_100_TE304_Offset				:	REAL;
H2SO4_PressureBeforeTubeReactor_100_Offset				:	REAL;
H3PO4_PressureBeforeTubeReactor_100_Offset				:	REAL;
AcidWaistPressure_100_Offset				:	REAL;
H2SO4_PressureBeforeTubeReactor_100_1_Offset				:	REAL;
H3PO4_PressureBeforeTubeReactor_100_1_Offset				:	REAL;
AcidWaistPressure_100_1_Offset				:	REAL;
H2SO4ConsumTubeReactor_100_Offset				:	REAL;
FCV3Pos_Offset				:	REAL;
H3PO4ConsumTubeReactor_100_Offset				:	REAL;
FCV4Pos_Offset				:	REAL;
AcidWaistConsume_100_Offset				:	REAL;
FCV5Pos_Offset				:	REAL;
FCV10Pos_Offset				:	REAL;
FCV214Pos_Offset				:	REAL;
FCV341Pos_Offset				:	REAL;
FCV342Pos_Offset				:	REAL;
H2SO4ConsumTubeReactor_100_1_Offset				:	REAL;
FCV343Pos_Offset				:	REAL;
H3PO4ConsumTubeReactor_100_1_Offset				:	REAL;
FCV344Pos_Offset				:	REAL;
AcidWaistConsume_100_1_Offset				:	REAL;
FCV345Pos_Offset				:	REAL;
FCV346Pos_Offset				:	REAL;
AntiCackLevelInReceivTank_81_Offset				:	REAL;
AntiCackLevelInSupplyTank_82_Offset				:	REAL;
SubPumpCurrent_102_B_Offset				:	REAL;
SubPumpCurrent_103_1B_Offset				:	REAL;



END_VAR

// Application/PLC_PRG
PROGRAM PLC_PRG
VAR
END_VAR

;

END_PROGRAM

// Application/IO/AI_TO_Current
FUNCTION AI_TO_Current : REAL
VAR_INPUT
	AI_Input	: INT;
END_VAR
VAR
END_VAR

AI_TO_Current:= ((TO_REAL(AI_Input))/32762) * 19.6 + 0.4;

END_FUNCTION

// Application/IO/prAItoValue
PROGRAM prAItoValue
VAR
END_VAR

TgasBeforeDryerDrum_45:= AI_TO_Current(AI_TgasBeforeDryerDrum_45) * TgasBeforeDryerDrum_45_CalCoef + TgasBeforeDryerDrum_45_Offset;
TgasAfterDryerDrum_45:= AI_TO_Current(AI_TgasAfterDryerDrum_45) * TgasAfterDryerDrum_45_CalCoef + TgasAfterDryerDrum_45_Offset;
TgasFurnace_120:= AI_TO_Current(AI_TgasFurnace_120) * TgasFurnace_120_CalCoef + TgasFurnace_120_Offset;
TproductAfterDryerDrum_45:= AI_TO_Current(AI_TproductAfterDryerDrum_45) * TproductAfterDryerDrum_45_CalCoef + TproductAfterDryerDrum_45_Offset;
TairCooler:= AI_TO_Current(AI_TairCooler) * TairCooler_CalCoef + TairCooler_Offset;
TairAfterDrumCond_76:= AI_TO_Current(AI_TairAfterDrumCond_76) * TairAfterDrumCond_76_CalCoef + TairAfterDrumCond_76_Offset;
Tvent_53_3_1:= AI_TO_Current(AI_Tvent_53_3_1) * Tvent_53_3_1_CalCoef + Tvent_53_3_1_Offset;
Tvent_53_3_2:= AI_TO_Current(AI_Tvent_53_3_2) * Tvent_53_3_2_CalCoef + Tvent_53_3_2_Offset;
Tvent_53_2_1:= AI_TO_Current(AI_Tvent_53_2_1) * Tvent_53_2_1_CalCoef + Tvent_53_2_1_Offset;
Tvent_53_2_2:= AI_TO_Current(AI_Tvent_53_2_2) * Tvent_53_2_2_CalCoef + Tvent_53_2_2_Offset;
Tvent_53_1_1:= AI_TO_Current(AI_Tvent_53_1_1) * Tvent_53_1_1_CalCoef + Tvent_53_1_1_Offset;
Tvent_53_1_2:= AI_TO_Current(AI_Tvent_53_1_2) * Tvent_53_1_2_CalCoef + Tvent_53_1_2_Offset;
Tvent_65_0_1:= AI_TO_Current(AI_Tvent_65_0_1) * Tvent_65_0_1_CalCoef + Tvent_65_0_1_Offset;
Tvent_65_0_2:= AI_TO_Current(AI_Tvent_65_0_2) * Tvent_65_0_2_CalCoef + Tvent_65_0_2_Offset;
Tvent_65_1_1:= AI_TO_Current(AI_Tvent_65_1_1) * Tvent_65_1_1_CalCoef + Tvent_65_1_1_Offset;
Tvent_65_1_2:= AI_TO_Current(AI_Tvent_65_1_2) * Tvent_65_1_2_CalCoef + Tvent_65_1_2_Offset;
Tvent_65_2_1:= AI_TO_Current(AI_Tvent_65_2_1) * Tvent_65_2_1_CalCoef + Tvent_65_2_1_Offset;
Tvent_65_2_2:= AI_TO_Current(AI_Tvent_65_2_2) * Tvent_65_2_2_CalCoef + Tvent_65_2_2_Offset;
Tretur_61:= AI_TO_Current(AI_Tretur_61) * Tretur_61_CalCoef + Tretur_61_Offset;
Ttank_103_1:= AI_TO_Current(AI_Ttank_103_1) * Ttank_103_1_CalCoef + Ttank_103_1_Offset;
AirPressureBeforeBurner:= AI_TO_Current(AI_AirPressureBeforeBurner) * AirPressureBeforeBurner_CalCoef + AirPressureBeforeBurner_Offset;
AirFirstPressureBeforeFurnace_120:= AI_TO_Current(AI_AirFirstPressureBeforeFurnace_120) * AirFirstPressureBeforeFurnace_120_CalCoef + AirFirstPressureBeforeFurnace_120_Offset;
AirSecondPressureBeforeFurnace_120:= AI_TO_Current(AI_AirSecondPressureBeforeFurnace_120) * AirSecondPressureBeforeFurnace_120_CalCoef + AirSecondPressureBeforeFurnace_120_Offset;
PCV22Pos:= AI_TO_Current(AI_PCV22Pos) * PCV22Pos_CalCoef + PCV22Pos_Offset;
UnderPresFurnace_120:= AI_TO_Current(AI_UnderPresFurnace_120) * UnderPresFurnace_120_CalCoef + UnderPresFurnace_120_Offset;
UnderPresGranul_31:= AI_TO_Current(AI_UnderPresGranul_31) * UnderPresGranul_31_CalCoef + UnderPresGranul_31_Offset;
UnderPresDryerDrum_45:= AI_TO_Current(AI_UnderPresDryerDrum_45) * UnderPresDryerDrum_45_CalCoef + UnderPresDryerDrum_45_Offset;
UnderPresCooler_63_1:= AI_TO_Current(AI_UnderPresCooler_63_1) * UnderPresCooler_63_1_CalCoef + UnderPresCooler_63_1_Offset;
PressureKiPA:= AI_TO_Current(AI_PressureKiPA) * PressureKiPA_CalCoef + PressureKiPA_Offset;
UnderPresBeforeAbsorbAKT_37:= AI_TO_Current(AI_UnderPresBeforeAbsorbAKT_37) * UnderPresBeforeAbsorbAKT_37_CalCoef + UnderPresBeforeAbsorbAKT_37_Offset;
UnderPresAfterAbsorbAKT_37:= AI_TO_Current(AI_UnderPresAfterAbsorbAKT_37) * UnderPresAfterAbsorbAKT_37_CalCoef + UnderPresAfterAbsorbAKT_37_Offset;
UnderPresAfterAPS_48:= AI_TO_Current(AI_UnderPresAfterAPS_48) * UnderPresAfterAPS_48_CalCoef + UnderPresAfterAPS_48_Offset;
UnderPresBeforeHydroCycl_21:= AI_TO_Current(AI_UnderPresBeforeHydroCycl_21) * UnderPresBeforeHydroCycl_21_CalCoef + UnderPresBeforeHydroCycl_21_Offset;
UnderPresAfterHydroCycl_21:= AI_TO_Current(AI_UnderPresAfterHydroCycl_21) * UnderPresAfterHydroCycl_21_CalCoef + UnderPresAfterHydroCycl_21_Offset;
UnderPresSalex_211:= AI_TO_Current(AI_UnderPresSalex_211) * UnderPresSalex_211_CalCoef + UnderPresSalex_211_Offset;
AbsorbConsumInHydroCycl_21:= AI_TO_Current(AI_AbsorbConsumInHydroCycl_21) * AbsorbConsumInHydroCycl_21_CalCoef + AbsorbConsumInHydroCycl_21_Offset;
AbsorbConsumBeforeHydroCycl_21:= AI_TO_Current(AI_AbsorbConsumBeforeHydroCycl_21) * AbsorbConsumBeforeHydroCycl_21_CalCoef + AbsorbConsumBeforeHydroCycl_21_Offset;
GasConsumBeforeBurner:= AI_TO_Current(AI_GasConsumBeforeBurner) * GasConsumBeforeBurner_CalCoef + GasConsumBeforeBurner_Offset;
FCV16Pos:= AI_TO_Current(AI_FCV16Pos) * FCV16Pos_CalCoef + FCV16Pos_Offset;
AirConsumeFurnace_120:= AI_TO_Current(AI_AirConsumeFurnace_120) * AirConsumeFurnace_120_CalCoef + AirConsumeFurnace_120_Offset;
FCV18Pos:= AI_TO_Current(AI_FCV18Pos) * FCV18Pos_CalCoef + FCV18Pos_Offset;
ReturConsumGranul_31:= AI_TO_Current(AI_ReturConsumGranul_31) * ReturConsumGranul_31_CalCoef + ReturConsumGranul_31_Offset;
AbsorLiquidConsumbAKT_37_FT100:= AI_TO_Current(AI_AbsorLiquidConsumbAKT_37_FT100) * AbsorLiquidConsumbAKT_37_FT100_CalCoef + AbsorLiquidConsumbAKT_37_FT100_Offset;
WaterConsumAbsorbSystem:= AI_TO_Current(AI_WaterConsumAbsorbSystem) * WaterConsumAbsorbSystem_CalCoef + WaterConsumAbsorbSystem_Offset;
AbsorLiquidScuber_66_12:= AI_TO_Current(AI_AbsorLiquidScuber_66_12) * AbsorLiquidScuber_66_12_CalCoef + AbsorLiquidScuber_66_12_Offset;
AbsorLiquidTank_103_1:= AI_TO_Current(AI_AbsorLiquidTank_103_1) * AbsorLiquidTank_103_1_CalCoef + AbsorLiquidTank_103_1_Offset;
FCV113:= AI_TO_Current(AI_FCV113) * FCV113_CalCoef + FCV113_Offset;
ConsumBeforeScrubber_66_1:= AI_TO_Current(AI_ConsumBeforeScrubber_66_1) * ConsumBeforeScrubber_66_1_CalCoef + ConsumBeforeScrubber_66_1_Offset;
ConsumInAPS_48:= AI_TO_Current(AI_ConsumInAPS_48) * ConsumInAPS_48_CalCoef + ConsumInAPS_48_Offset;
ConsumH2SO4_102_to_35:= AI_TO_Current(AI_ConsumH2SO4_102_to_35) * ConsumH2SO4_102_to_35_CalCoef + ConsumH2SO4_102_to_35_Offset;
ConsumH2SO4_102_to_103:= AI_TO_Current(AI_ConsumH2SO4_102_to_103) * ConsumH2SO4_102_to_103_CalCoef + ConsumH2SO4_102_to_103_Offset;
AbsorLiquidConsumbAKT_37_FT132:= AI_TO_Current(AI_AbsorLiquidConsumbAKT_37_FT132) * AbsorLiquidConsumbAKT_37_FT132_CalCoef + AbsorLiquidConsumbAKT_37_FT132_Offset;
Consum_H3PO4:= AI_TO_Current(AI_Consum_H3PO4) * Consum_H3PO4_CalCoef + Consum_H3PO4_Offset;
ConsumH2SO4:= AI_TO_Current(AI_ConsumH2SO4) * ConsumH2SO4_CalCoef + ConsumH2SO4_Offset;
ConsumPressedAirToZech:= AI_TO_Current(AI_ConsumPressedAirToZech) * ConsumPressedAirToZech_CalCoef + ConsumPressedAirToZech_Offset;
ConsumPressedAir:= AI_TO_Current(AI_ConsumPressedAir) * ConsumPressedAir_CalCoef + ConsumPressedAir_Offset;
ConsumChlKToGran_FQUIR_12_31:= AI_TO_Current(AI_ConsumChlKToGran_FQUIR_12_31) * ConsumChlKToGran_FQUIR_12_31_CalCoef + ConsumChlKToGran_FQUIR_12_31_Offset;
ConsumKarbanToGran_31:= AI_TO_Current(AI_ConsumKarbanToGran_31) * ConsumKarbanToGran_31_CalCoef + ConsumKarbanToGran_31_Offset;
ConsumChlKToGran_FQUIR_17_31:= AI_TO_Current(AI_ConsumChlKToGran_FQUIR_17_31) * ConsumChlKToGran_FQUIR_17_31_CalCoef + ConsumChlKToGran_FQUIR_17_31_Offset;
ConsumMicroAddToGran_31_FQUIR_57_1:= AI_TO_Current(AI_ConsumMicroAddToGran_31_FQUIR_57_1) * ConsumMicroAddToGran_31_FQUIR_57_1_CalCoef + ConsumMicroAddToGran_31_FQUIR_57_1_Offset;
ConsumMicroAddToGran_31_FQUIR_57_2:= AI_TO_Current(AI_ConsumMicroAddToGran_31_FQUIR_57_2) * ConsumMicroAddToGran_31_FQUIR_57_2_CalCoef + ConsumMicroAddToGran_31_FQUIR_57_2_Offset;
OilLevel_78:= AI_TO_Current(AI_OilLevel_78) * OilLevel_78_CalCoef + OilLevel_78_Offset;
CycleTankLevel_49:= AI_TO_Current(AI_CycleTankLevel_49) * CycleTankLevel_49_CalCoef + CycleTankLevel_49_Offset;
LCV101Pos:= AI_TO_Current(AI_LCV101Pos) * LCV101Pos_CalCoef + LCV101Pos_Offset;
CollectorTankLevel_35:= AI_TO_Current(AI_CollectorTankLevel_35) * CollectorTankLevel_35_CalCoef + CollectorTankLevel_35_Offset;
CycleTankLevel_67:= AI_TO_Current(AI_CycleTankLevel_67) * CycleTankLevel_67_CalCoef + CycleTankLevel_67_Offset;
CollectorTankLevel_103_1:= AI_TO_Current(AI_CollectorTankLevel_103_1) * CollectorTankLevel_103_1_CalCoef + CollectorTankLevel_103_1_Offset;
ReceivTankH3PO4level_41:= AI_TO_Current(AI_ReceivTankH3PO4level_41) * ReceivTankH3PO4level_41_CalCoef + ReceivTankH3PO4level_41_Offset;
ReceivTankH3PO4level_39:= AI_TO_Current(AI_ReceivTankH3PO4level_39) * ReceivTankH3PO4level_39_CalCoef + ReceivTankH3PO4level_39_Offset;
SupplyTankH3PO4level_25:= AI_TO_Current(AI_SupplyTankH3PO4level_25) * SupplyTankH3PO4level_25_CalCoef + SupplyTankH3PO4level_25_Offset;
LCV203Pos:= AI_TO_Current(AI_LCV203Pos) * LCV203Pos_CalCoef + LCV203Pos_Offset;
TankH2SO4Level_102:= AI_TO_Current(AI_TankH2SO4Level_102) * TankH2SO4Level_102_CalCoef + TankH2SO4Level_102_Offset;
SupplyTankH2SO4Level_102_a:= AI_TO_Current(AI_SupplyTankH2SO4Level_102_a) * SupplyTankH2SO4Level_102_a_CalCoef + SupplyTankH2SO4Level_102_a_Offset;
LCV206Pos:= AI_TO_Current(AI_LCV206Pos) * LCV206Pos_CalCoef + LCV206Pos_Offset;
pH_CollectorTank_35:= AI_TO_Current(AI_pH_CollectorTank_35) * pH_CollectorTank_35_CalCoef + pH_CollectorTank_35_Offset;
ACV104Pos:= AI_TO_Current(AI_ACV104Pos) * ACV104Pos_CalCoef + ACV104Pos_Offset;
pH_CyclTank_49:= AI_TO_Current(AI_pH_CyclTank_49) * pH_CyclTank_49_CalCoef + pH_CyclTank_49_Offset;
ACV112Pos:= AI_TO_Current(AI_ACV112Pos) * ACV112Pos_CalCoef + ACV112Pos_Offset;
pH_CollectorTank_103_1:= AI_TO_Current(AI_pH_CollectorTank_103_1) * pH_CollectorTank_103_1_CalCoef + pH_CollectorTank_103_1_Offset;
ACV115Pos:= AI_TO_Current(AI_ACV115Pos) * ACV115Pos_CalCoef + ACV115Pos_Offset;
OutAirWetness:= AI_TO_Current(AI_OutAirWetness) * OutAirWetness_CalCoef + OutAirWetness_Offset;
DryerRoomAirWetness_45:= AI_TO_Current(AI_DryerRoomAirWetness_45) * DryerRoomAirWetness_45_CalCoef + DryerRoomAirWetness_45_Offset;
IssuedProductWeight_203:= AI_TO_Current(AI_IssuedProductWeight_203) * IssuedProductWeight_203_CalCoef + IssuedProductWeight_203_Offset;
TubeReactorTemp_100_TE9:= AI_TO_Current(AI_TubeReactorTemp_100_TE9) * TubeReactorTemp_100_TE9_CalCoef + TubeReactorTemp_100_TE9_Offset;
AntiCackTempInReceiveTank_81:= AI_TO_Current(AI_AntiCackTempInReceiveTank_81) * AntiCackTempInReceiveTank_81_CalCoef + AntiCackTempInReceiveTank_81_Offset;
TCV302Pos:= AI_TO_Current(AI_TCV302Pos) * TCV302Pos_CalCoef + TCV302Pos_Offset;
AntiCackTempInSupplyTank_81_TT303:= AI_TO_Current(AI_AntiCackTempInSupplyTank_81_TT303) * AntiCackTempInSupplyTank_81_TT303_CalCoef + AntiCackTempInSupplyTank_81_TT303_Offset;
TCV303Pos:= AI_TO_Current(AI_TCV303Pos) * TCV303Pos_CalCoef + TCV303Pos_Offset;
TubeReactorTemp_100_TE304:= AI_TO_Current(AI_TubeReactorTemp_100_TE304) * TubeReactorTemp_100_TE304_CalCoef + TubeReactorTemp_100_TE304_Offset;
H2SO4_PressureBeforeTubeReactor_100:= AI_TO_Current(AI_H2SO4_PressureBeforeTubeReactor_100) * H2SO4_PressureBeforeTubeReactor_100_CalCoef + H2SO4_PressureBeforeTubeReactor_100_Offset;
H3PO4_PressureBeforeTubeReactor_100:= AI_TO_Current(AI_H3PO4_PressureBeforeTubeReactor_100) * H3PO4_PressureBeforeTubeReactor_100_CalCoef + H3PO4_PressureBeforeTubeReactor_100_Offset;
AcidWaistPressure_100:= AI_TO_Current(AI_AcidWaistPressure_100) * AcidWaistPressure_100_CalCoef + AcidWaistPressure_100_Offset;
H2SO4_PressureBeforeTubeReactor_100_1:= AI_TO_Current(AI_H2SO4_PressureBeforeTubeReactor_100_1) * H2SO4_PressureBeforeTubeReactor_100_1_CalCoef + H2SO4_PressureBeforeTubeReactor_100_1_Offset;
H3PO4_PressureBeforeTubeReactor_100_1:= AI_TO_Current(AI_H3PO4_PressureBeforeTubeReactor_100_1) * H3PO4_PressureBeforeTubeReactor_100_1_CalCoef + H3PO4_PressureBeforeTubeReactor_100_1_Offset;
AcidWaistPressure_100_1:= AI_TO_Current(AI_AcidWaistPressure_100_1) * AcidWaistPressure_100_1_CalCoef + AcidWaistPressure_100_1_Offset;
H2SO4ConsumTubeReactor_100:= AI_TO_Current(AI_H2SO4ConsumTubeReactor_100) * H2SO4ConsumTubeReactor_100_CalCoef + H2SO4ConsumTubeReactor_100_Offset;
FCV3Pos:= AI_TO_Current(AI_FCV3Pos) * FCV3Pos_CalCoef + FCV3Pos_Offset;
H3PO4ConsumTubeReactor_100:= AI_TO_Current(AI_H3PO4ConsumTubeReactor_100) * H3PO4ConsumTubeReactor_100_CalCoef + H3PO4ConsumTubeReactor_100_Offset;
FCV4Pos:= AI_TO_Current(AI_FCV4Pos) * FCV4Pos_CalCoef + FCV4Pos_Offset;
AcidWaistConsume_100:= AI_TO_Current(AI_AcidWaistConsume_100) * AcidWaistConsume_100_CalCoef + AcidWaistConsume_100_Offset;
FCV5Pos:= AI_TO_Current(AI_FCV5Pos) * FCV5Pos_CalCoef + FCV5Pos_Offset;
FCV10Pos:= AI_TO_Current(AI_FCV10Pos) * FCV10Pos_CalCoef + FCV10Pos_Offset;
FCV214Pos:= AI_TO_Current(AI_FCV214Pos) * FCV214Pos_CalCoef + FCV214Pos_Offset;
FCV341Pos:= AI_TO_Current(AI_FCV341Pos) * FCV341Pos_CalCoef + FCV341Pos_Offset;
FCV342Pos:= AI_TO_Current(AI_FCV342Pos) * FCV342Pos_CalCoef + FCV342Pos_Offset;
H2SO4ConsumTubeReactor_100_1:= AI_TO_Current(AI_H2SO4ConsumTubeReactor_100_1) * H2SO4ConsumTubeReactor_100_1_CalCoef + H2SO4ConsumTubeReactor_100_1_Offset;
FCV343Pos:= AI_TO_Current(AI_FCV343Pos) * FCV343Pos_CalCoef + FCV343Pos_Offset;
H3PO4ConsumTubeReactor_100_1:= AI_TO_Current(AI_H3PO4ConsumTubeReactor_100_1) * H3PO4ConsumTubeReactor_100_1_CalCoef + H3PO4ConsumTubeReactor_100_1_Offset;
FCV344Pos:= AI_TO_Current(AI_FCV344Pos) * FCV344Pos_CalCoef + FCV344Pos_Offset;
AcidWaistConsume_100_1:= AI_TO_Current(AI_AcidWaistConsume_100_1) * AcidWaistConsume_100_1_CalCoef + AcidWaistConsume_100_1_Offset;
FCV345Pos:= AI_TO_Current(AI_FCV345Pos) * FCV345Pos_CalCoef + FCV345Pos_Offset;
FCV346Pos:= AI_TO_Current(AI_FCV346Pos) * FCV346Pos_CalCoef + FCV346Pos_Offset;
AntiCackLevelInReceivTank_81:= AI_TO_Current(AI_AntiCackLevelInReceivTank_81) * AntiCackLevelInReceivTank_81_CalCoef + AntiCackLevelInReceivTank_81_Offset;
AntiCackLevelInSupplyTank_82:= AI_TO_Current(AI_AntiCackLevelInSupplyTank_82) * AntiCackLevelInSupplyTank_82_CalCoef + AntiCackLevelInSupplyTank_82_Offset;
SubPumpCurrent_102_B:= AI_TO_Current(AI_SubPumpCurrent_102_B) * SubPumpCurrent_102_B_CalCoef + SubPumpCurrent_102_B_Offset;
SubPumpCurrent_103_1B:= AI_TO_Current(AI_SubPumpCurrent_103_1B) * SubPumpCurrent_103_1B_CalCoef + SubPumpCurrent_103_1B_Offset;

END_PROGRAM

// Application/IO/prInToVars
PROGRAM prInToVars
VAR
END_VAR

DI_GasFurnaceMinLevelAlm	:=	_DI_GasFurnaceMinLevelAlm	;
DI_BunkerMaxLevel_88_2	:=	_DI_BunkerMaxLevel_88_2	;
DI_BunkerMaxLevel_88_1	:=	_DI_BunkerMaxLevel_88_1	;
DI_BunkerMaxLevel_70_1	:=	_DI_BunkerMaxLevel_70_1	;
DI_BunkerMaxLevel_70_2	:=	_DI_BunkerMaxLevel_70_2	;
DI_BunkerMaxLevel_86	:=	_DI_BunkerMaxLevel_86	;
DI_ElevatorMaxLevel_54	:=	_DI_ElevatorMaxLevel_54	;
DI_OvenMaxLevel_58_1	:=	_DI_OvenMaxLevel_58_1	;
DI_ElevatorMaxLevel_214_1	:=	_DI_ElevatorMaxLevel_214_1	;
DI_MainBurnerFire_120	:=	_DI_MainBurnerFire_120	;
DI_IgnitionBurnerFire_120	:=	_DI_IgnitionBurnerFire_120	;
DI_SupplierMotorWork_57_1	:=	_DI_SupplierMotorWork_57_1	;
DI_SupplierMotorAlm_57_1	:=	_DI_SupplierMotorAlm_57_1	;
DI_SupplierMotorWork_57_2	:=	_DI_SupplierMotorWork_57_2	;
DI_SupplierMotorAlm_57_2	:=	_DI_SupplierMotorAlm_57_2	;
DI_SupplierMotorWork_71_1	:=	_DI_SupplierMotorWork_71_1	;
DI_SupplierMotorAlm_71_1	:=	_DI_SupplierMotorAlm_71_1	;
DI_SupplierMotorWork_71_2	:=	_DI_SupplierMotorWork_71_2	;
DI_SupplierMotorAlm_71_2	:=	_DI_SupplierMotorAlm_71_2	;
DI_SupplierMotorWork_87_1	:=	_DI_SupplierMotorWork_87_1	;
DI_SupplierMotorAlm_87_1	:=	_DI_SupplierMotorAlm_87_1	;
DI_DryerDrumMotorNotWorking_45_53	:=	_DI_DryerDrumMotorNotWorking_45_53	;
DI_UPS_Bypass_1	:=	_DI_UPS_Bypass_1	;
DI_UPS_Battery_1	:=	_DI_UPS_Battery_1	;
DI_UPS_BatteryDischarge_1	:=	_DI_UPS_BatteryDischarge_1	;
DI_UPS_Alm_1	:=	_DI_UPS_Alm_1	;
DI_UPS_Bypass_2	:=	_DI_UPS_Bypass_2	;
DI_UPS_Battery_2	:=	_DI_UPS_Battery_2	;
DI_UPS_BatteryDischarge_2	:=	_DI_UPS_BatteryDischarge_2	;
DI_UPS_Alm_2	:=	_DI_UPS_Alm_2	;
DI_PowerRackVoltageOn_1	:=	_DI_PowerRackVoltageOn_1	;
DI_PowerRackVoltageOn_2	:=	_DI_PowerRackVoltageOn_2	;
DI_PowerRackAlmStop_1	:=	_DI_PowerRackAlmStop_1	;
DI_PowerRackAlmStop_2	:=	_DI_PowerRackAlmStop_2	;
DI_SubPumpWorking_25_1B	:=	_DI_SubPumpWorking_25_1B	;
DI_AntiCackPumpWorking_81_1	:=	_DI_AntiCackPumpWorking_81_1	;
DI_AntiCackPumpWorking_81_2	:=	_DI_AntiCackPumpWorking_81_2	;
DI_AntiCackPumpWorking_82_1	:=	_DI_AntiCackPumpWorking_82_1	;
DI_AntiCackPumpWorking_82_2	:=	_DI_AntiCackPumpWorking_82_2	;
DI_SubPumpWorking_102_B	:=	_DI_SubPumpWorking_102_B	;

///////////////////////////////////////////////////////////////////////////////////////////////////////



AI_TgasBeforeDryerDrum_45	:=	_AI_TgasBeforeDryerDrum_45	;
AI_TgasAfterDryerDrum_45	:=	_AI_TgasAfterDryerDrum_45	;
AI_TgasFurnace_120	:=	_AI_TgasFurnace_120	;
AI_TproductAfterDryerDrum_45	:=	_AI_TproductAfterDryerDrum_45	;
AI_TairCooler	:=	_AI_TairCooler	;
AI_TairAfterDrumCond_76	:=	_AI_TairAfterDrumCond_76	;
AI_Tvent_53_3_1	:=	_AI_Tvent_53_3_1	;
AI_Tvent_53_3_2	:=	_AI_Tvent_53_3_2	;
AI_Tvent_53_2_1	:=	_AI_Tvent_53_2_1	;
AI_Tvent_53_2_2	:=	_AI_Tvent_53_2_2	;
AI_Tvent_53_1_1	:=	_AI_Tvent_53_1_1	;
AI_Tvent_53_1_2	:=	_AI_Tvent_53_1_2	;
AI_Tvent_65_0_1	:=	_AI_Tvent_65_0_1	;
AI_Tvent_65_0_2	:=	_AI_Tvent_65_0_2	;
AI_Tvent_65_1_1	:=	_AI_Tvent_65_1_1	;
AI_Tvent_65_1_2	:=	_AI_Tvent_65_1_2	;
AI_Tvent_65_2_1	:=	_AI_Tvent_65_2_1	;
AI_Tvent_65_2_2	:=	_AI_Tvent_65_2_2	;
AI_Tretur_61	:=	_AI_Tretur_61	;
AI_Ttank_103_1	:=	_AI_Ttank_103_1	;
AI_AirPressureBeforeBurner	:=	_AI_AirPressureBeforeBurner	;
AI_AirFirstPressureBeforeFurnace_120	:=	_AI_AirFirstPressureBeforeFurnace_120	;
AI_AirSecondPressureBeforeFurnace_120	:=	_AI_AirSecondPressureBeforeFurnace_120	;
AI_PCV22Pos	:=	_AI_PCV22Pos	;
AI_UnderPresFurnace_120	:=	_AI_UnderPresFurnace_120	;
AI_UnderPresGranul_31	:=	_AI_UnderPresGranul_31	;
AI_UnderPresDryerDrum_45	:=	_AI_UnderPresDryerDrum_45	;
AI_UnderPresCooler_63_1	:=	_AI_UnderPresCooler_63_1	;
AI_PressureKiPA	:=	_AI_PressureKiPA	;
AI_UnderPresBeforeAbsorbAKT_37	:=	_AI_UnderPresBeforeAbsorbAKT_37	;
AI_UnderPresAfterAbsorbAKT_37	:=	_AI_UnderPresAfterAbsorbAKT_37	;
AI_UnderPresAfterAPS_48	:=	_AI_UnderPresAfterAPS_48	;
AI_UnderPresBeforeHydroCycl_21	:=	_AI_UnderPresBeforeHydroCycl_21	;
AI_UnderPresAfterHydroCycl_21	:=	_AI_UnderPresAfterHydroCycl_21	;
AI_UnderPresSalex_211	:=	_AI_UnderPresSalex_211	;
AI_AbsorbConsumInHydroCycl_21	:=	_AI_AbsorbConsumInHydroCycl_21	;
AI_AbsorbConsumBeforeHydroCycl_21	:=	_AI_AbsorbConsumBeforeHydroCycl_21	;
AI_GasConsumBeforeBurner	:=	_AI_GasConsumBeforeBurner	;
AI_FCV16Pos	:=	_AI_FCV16Pos	;
AI_AirConsumeFurnace_120	:=	_AI_AirConsumeFurnace_120	;
AI_FCV18Pos	:=	_AI_FCV18Pos	;
AI_ReturConsumGranul_31	:=	_AI_ReturConsumGranul_31	;
AI_AbsorLiquidConsumbAKT_37_FT100	:=	_AI_AbsorLiquidConsumbAKT_37_FT100	;
AI_WaterConsumAbsorbSystem	:=	_AI_WaterConsumAbsorbSystem	;
AI_AbsorLiquidScuber_66_12	:=	_AI_AbsorLiquidScuber_66_12	;
AI_AbsorLiquidTank_103_1	:=	_AI_AbsorLiquidTank_103_1	;
AI_FCV113	:=	_AI_FCV113	;
AI_ConsumBeforeScrubber_66_1	:=	_AI_ConsumBeforeScrubber_66_1	;
AI_ConsumInAPS_48	:=	_AI_ConsumInAPS_48	;
AI_ConsumH2SO4_102_to_35	:=	_AI_ConsumH2SO4_102_to_35	;
AI_ConsumH2SO4_102_to_103	:=	_AI_ConsumH2SO4_102_to_103	;
AI_AbsorLiquidConsumbAKT_37_FT132	:=	_AI_AbsorLiquidConsumbAKT_37_FT132	;
AI_Consum_H3PO4	:=	_AI_Consum_H3PO4	;
AI_ConsumH2SO4	:=	_AI_ConsumH2SO4	;
AI_ConsumPressedAirToZech	:=	_AI_ConsumPressedAirToZech	;
AI_ConsumPressedAir	:=	_AI_ConsumPressedAir	;
AI_ConsumChlKToGran_FQUIR_12_31	:=	_AI_ConsumChlKToGran_FQUIR_12_31	;
AI_ConsumKarbanToGran_31	:=	_AI_ConsumKarbanToGran_31	;
AI_ConsumChlKToGran_FQUIR_17_31	:=	_AI_ConsumChlKToGran_FQUIR_17_31	;
AI_ConsumMicroAddToGran_31_FQUIR_57_1	:=	_AI_ConsumMicroAddToGran_31_FQUIR_57_1	;
AI_ConsumMicroAddToGran_31_FQUIR_57_2	:=	_AI_ConsumMicroAddToGran_31_FQUIR_57_2	;
AI_OilLevel_78	:=	_AI_OilLevel_78	;
AI_CycleTankLevel_49	:=	_AI_CycleTankLevel_49	;
AI_LCV101Pos	:=	_AI_LCV101Pos	;
AI_CollectorTankLevel_35	:=	_AI_CollectorTankLevel_35	;
AI_CycleTankLevel_67	:=	_AI_CycleTankLevel_67	;
AI_CollectorTankLevel_103_1	:=	_AI_CollectorTankLevel_103_1	;
AI_ReceivTankH3PO4level_41	:=	_AI_ReceivTankH3PO4level_41	;
AI_ReceivTankH3PO4level_39	:=	_AI_ReceivTankH3PO4level_39	;
AI_SupplyTankH3PO4level_25	:=	_AI_SupplyTankH3PO4level_25	;
AI_LCV203Pos	:=	_AI_LCV203Pos	;
AI_TankH2SO4Level_102	:=	_AI_TankH2SO4Level_102	;
AI_SupplyTankH2SO4Level_102_a	:=	_AI_SupplyTankH2SO4Level_102_a	;
AI_LCV206Pos	:=	_AI_LCV206Pos	;
AI_pH_CollectorTank_35	:=	_AI_pH_CollectorTank_35	;
AI_ACV104Pos	:=	_AI_ACV104Pos	;
AI_pH_CyclTank_49	:=	_AI_pH_CyclTank_49	;
AI_ACV112Pos	:=	_AI_ACV112Pos	;
AI_pH_CollectorTank_103_1	:=	_AI_pH_CollectorTank_103_1	;
AI_ACV115Pos	:=	_AI_ACV115Pos	;
AI_OutAirWetness	:=	_AI_OutAirWetness	;
AI_DryerRoomAirWetness_45	:=	_AI_DryerRoomAirWetness_45	;
AI_IssuedProductWeight_203	:=	_AI_IssuedProductWeight_203	;
AI_TubeReactorTemp_100_TE9	:=	_AI_TubeReactorTemp_100_TE9	;
AI_AntiCackTempInReceiveTank_81	:=	_AI_AntiCackTempInReceiveTank_81	;
AI_TCV302Pos	:=	_AI_TCV302Pos	;
AI_AntiCackTempInSupplyTank_81_TT303	:=	_AI_AntiCackTempInSupplyTank_81_TT303	;
AI_TCV303Pos	:=	_AI_TCV303Pos	;
AI_TubeReactorTemp_100_TE304	:=	_AI_TubeReactorTemp_100_TE304	;
AI_H2SO4_PressureBeforeTubeReactor_100	:=	_AI_H2SO4_PressureBeforeTubeReactor_100	;
AI_H3PO4_PressureBeforeTubeReactor_100	:=	_AI_H3PO4_PressureBeforeTubeReactor_100	;
AI_AcidWaistPressure_100	:=	_AI_AcidWaistPressure_100	;
AI_H2SO4_PressureBeforeTubeReactor_100_1	:=	_AI_H2SO4_PressureBeforeTubeReactor_100_1	;
AI_H3PO4_PressureBeforeTubeReactor_100_1	:=	_AI_H3PO4_PressureBeforeTubeReactor_100_1	;
AI_AcidWaistPressure_100_1	:=	_AI_AcidWaistPressure_100_1	;
AI_H2SO4ConsumTubeReactor_100	:=	_AI_H2SO4ConsumTubeReactor_100	;
AI_FCV3Pos	:=	_AI_FCV3Pos	;
AI_H3PO4ConsumTubeReactor_100	:=	_AI_H3PO4ConsumTubeReactor_100	;
AI_FCV4Pos	:=	_AI_FCV4Pos	;
AI_AcidWaistConsume_100	:=	_AI_AcidWaistConsume_100	;
AI_FCV5Pos	:=	_AI_FCV5Pos	;
AI_FCV10Pos	:=	_AI_FCV10Pos	;
AI_FCV214Pos	:=	_AI_FCV214Pos	;
AI_FCV341Pos	:=	_AI_FCV341Pos	;
AI_FCV342Pos	:=	_AI_FCV342Pos	;
AI_H2SO4ConsumTubeReactor_100_1	:=	_AI_H2SO4ConsumTubeReactor_100_1	;
AI_FCV343Pos	:=	_AI_FCV343Pos	;
AI_H3PO4ConsumTubeReactor_100_1	:=	_AI_H3PO4ConsumTubeReactor_100_1	;
AI_FCV344Pos	:=	_AI_FCV344Pos	;
AI_AcidWaistConsume_100_1	:=	_AI_AcidWaistConsume_100_1	;
AI_FCV345Pos	:=	_AI_FCV345Pos	;
AI_FCV346Pos	:=	_AI_FCV346Pos	;
AI_AntiCackLevelInReceivTank_81	:=	_AI_AntiCackLevelInReceivTank_81	;
AI_AntiCackLevelInSupplyTank_82	:=	_AI_AntiCackLevelInSupplyTank_82	;
AI_SubPumpCurrent_102_B	:=	_AI_SubPumpCurrent_102_B	;
AI_SubPumpCurrent_103_1B	:=	_AI_SubPumpCurrent_103_1B	;

END_PROGRAM

// Application/IO/prVarsToOut
PROGRAM prVarsToOut
VAR
END_VAR

_DO_SupplyStart_57_1	:=	DO_SupplyStart_57_1	;
_DO_SupplyStop_57_1	:=	DO_SupplyStop_57_1	;
_DO_SupplyStart_57_2	:=	DO_SupplyStart_57_2	;
_DO_SupplyStop_57_2	:=	DO_SupplyStop_57_2	;
_DO_SupplyStart_71_1	:=	DO_SupplyStart_71_1	;
_DO_SupplyStop_71_1	:=	DO_SupplyStop_71_1	;
_DO_SupplyStart_71_2	:=	DO_SupplyStart_71_2	;
_DO_SupplyStop_71_2	:=	DO_SupplyStop_71_2	;
_DO_SupplyStart_81_1	:=	DO_SupplyStart_81_1	;
_DO_SupplyStop_81_1	:=	DO_SupplyStop_81_1	;
_DO_MaxLevel_70_1_70_2_Stp_Elv8_Cvr5_6A	:=	DO_MaxLevel_70_1_70_2_Stp_Elv8_Cvr5_6A	;
_DO_MaxLevel_86_Stp_Elv8_Cvr5_7	:=	DO_MaxLevel_86_Stp_Elv8_Cvr5_7	;
_DO_MinLevel_49_Stp_Pump_50	:=	DO_MinLevel_49_Stp_Pump_50	;
_DO_MaxLevel_49_Stp_Pump_50	:=	DO_MaxLevel_49_Stp_Pump_50	;
_DO_MinLevel_67_Stp_Pump_68	:=	DO_MinLevel_67_Stp_Pump_68	;
_DO_MaxLevel_67_Stp_Pump_68	:=	DO_MaxLevel_67_Stp_Pump_68	;
_DO_MinLevel_67_Stp_Pump_68_1	:=	DO_MinLevel_67_Stp_Pump_68_1	;
_DO_MaxLevel_67_Stp_Pump_68_1	:=	DO_MaxLevel_67_Stp_Pump_68_1	;
_DO_MinLevel_103_1_Stp_Pump_103_1A	:=	DO_MinLevel_103_1_Stp_Pump_103_1A	;
_DO_MinLevelL1_103_1_Stp_Pump_103_1B	:=	DO_MinLevelL1_103_1_Stp_Pump_103_1B	;
_DO_MinLevelL2_103_1_Stp_Pump_103_1B	:=	DO_MinLevelL2_103_1_Stp_Pump_103_1B	;


///////////////////////////////////////////////////////////////////////////////////////////

_AO_AirPressureBeforeFenese_120	:=	AO_AirPressureBeforeFenese_120	;
_AO_GasFlowBeforeBurner	:=	AO_GasFlowBeforeBurner	;
_AO_AirFlowFenese_120	:=	AO_AirFlowFenese_120	;
_AO_AbsorbLiquidTo_103_1	:=	AO_AbsorbLiquidTo_103_1	;
_AO_ChlorKFlowToGranul_31_FQIR12	:=	AO_ChlorKFlowToGranul_31_FQIR12	;
_AO_KarbonFlowToGranul_31	:=	AO_KarbonFlowToGranul_31	;
_AO_ChlorKFlowToGranul_31_FQIR17	:=	AO_ChlorKFlowToGranul_31_FQIR17	;
_AO_MicroAddToGranul_31_FQIR57_1	:=	AO_MicroAddToGranul_31_FQIR57_1	;
_AO_MicroAddToGranul_31_FQIR57_2	:=	AO_MicroAddToGranul_31_FQIR57_2	;
_AO_SetLevelCyclTank_49	:=	AO_SetLevelCyclTank_49	;
_AO_SetLevelH3PO4SupplyTank_25	:=	AO_SetLevelH3PO4SupplyTank_25	;
_AO_SetLevelH2SO4SupplyTank_102_a	:=	AO_SetLevelH2SO4SupplyTank_102_a	;
_AO_Set_pHCollectTank_35	:=	AO_Set_pHCollectTank_35	;
_AO_Set_pHCycleTank_49	:=	AO_Set_pHCycleTank_49	;
_AO_Set_pHCollectTank_103_1	:=	AO_Set_pHCollectTank_103_1	;
_AO_SetShyberVent_53_3	:=	AO_SetShyberVent_53_3	;
_AO_SetShyberVent_53_2	:=	AO_SetShyberVent_53_2	;
_AO_SetShyberVent_53_1	:=	AO_SetShyberVent_53_1	;
_AO_SetShyberVent_65_0	:=	AO_SetShyberVent_65_0	;
_AO_SetShyberVent_65_1	:=	AO_SetShyberVent_65_1	;
_AO_SetShyberVent_65_2	:=	AO_SetShyberVent_65_2	;
_AO_SetAntiCackTempInCollectTank_81	:=	AO_SetAntiCackTempInCollectTank_81	;
_AO_SetAntiCackTempInCollectTank_82	:=	AO_SetAntiCackTempInCollectTank_82	;
_AO_SetH2SO4SupplyToTubeReactor_100	:=	AO_SetH2SO4SupplyToTubeReactor_100	;
_AO_SetH3PO4SupplyToTubeReactor_100	:=	AO_SetH3PO4SupplyToTubeReactor_100	;
_AO_SetAcidWaistFlowToTubeReactor_100	:=	AO_SetAcidWaistFlowToTubeReactor_100	;
_AO_SetNH3FlowToTubeReactor_100	:=	AO_SetNH3FlowToTubeReactor_100	;
_AO_SetSteamFlowToTubeReactor_100	:=	AO_SetSteamFlowToTubeReactor_100	;
_AO_SetAntiCackFlawToCondDrum_76	:=	AO_SetAntiCackFlawToCondDrum_76	;
_AO_SetNH3FlowToTubeReactor_100_1	:=	AO_SetNH3FlowToTubeReactor_100_1	;
_AO_SetH2SO4SupplyToTubeReactor_100_1	:=	AO_SetH2SO4SupplyToTubeReactor_100_1	;
_AO_SetH3PO4SupplyToTubeReactor_100_1	:=	AO_SetH3PO4SupplyToTubeReactor_100_1	;
_AO_SetAcidWaistFlowToTubeReactor_100_1	:=	AO_SetAcidWaistFlowToTubeReactor_100_1	;
_AO_SetSteamFlowToTubeReactor_100_1	:=	AO_SetSteamFlowToTubeReactor_100_1	;

END_PROGRAM
